PROGRAM MAIN
VAR
END_VAR

P_Strategy();

END_PROGRAM

(* stored: Version 1.1.0.1, ProductVersion 3.1.4024.12
   POU MAIN: Id {ec91c5d5-3c79-425d-bf90-5ff81ab84874}, SpecialFunc None *)
